# EPICS substitutions: respmat/respmatApp/Db/user.substitutions
# Example substitutions file

file "db/dbExample1.db" {
    { user = "lyyang" }
}

file db/dbExample2.db {
    pattern { user, no, scan }
        { "lyyang", 1, "1 second" }
        { "lyyang", 2, "2 second" }
        { "lyyang", 3, "5 second" }
}
